FUNCTION_BLOCK FB_AnalogLamp
VAR_INPUT
END_VAR
VAR_OUTPUT
END_VAR
VAR
END_VAR

END_FUNCTION_BLOCK

(* stored: Version 1.1.0.1, ProductVersion 3.1.4024.12
   POU FB_AnalogLamp: Id {6d09c337-7c6d-47a1-8e8a-78d8ffce0641}, SpecialFunc None *)
